{attribute 'qualified_only'}
{attribute 'strict'}
TYPE E_PositionState :
(
RETRACTED	:= 0,
INSERTED	:= 1,
MOVING	:= 2,
INVALID :=3
);
END_TYPE

(* stored: Version 1.1.0.1, ProductVersion 3.1.4022.18
   DUT E_PositionState: Id {580eeee3-6c52-42e6-b317-6ce95975b196} *)
